FUNCTION_BLOCK Current EXTENDS SM_Current
VAR_INPUT
END_VAR
VAR_OUTPUT
END_VAR
VAR
    _testVar : INT;
END_VAR

SUPER^();

END_FUNCTION_BLOCK

(* stored: Version 1.1.0.1, ProductVersion 3.1.4018.2
   POU Current: Id {486bf2a4-522c-4124-b0bc-3cc8c92a11ab}, SpecialFunc None *)
